PROGRAM MAIN
// Program başlangıç
VAR
    ButtonState : BOOL; // Buton durumu
    LampState : BOOL; // Lamba durumu
END_VAR

// Ana döngü

// Ana döngü
WHILE TRUE DO
    // Buton durumunu kontrol et
    ButtonState := ReadButtonState();

    // Buton basıldıysa
    IF ButtonState THEN
        // Lambayı aç
        LampState := TRUE;
    ELSE
        // Lambayı kapat
        LampState := FALSE;
    END_IF

END_PROGRAM

(* stored: Version 1.1.0.1, ProductVersion 3.1.4024.12
   POU MAIN: Id {ed56a81f-7398-444e-ad3f-188292cf87d3}, SpecialFunc None *)
